{attribute addProperty BoxType "EPP3744-0041-0016"}
{attribute addProperty Id "Safe_State_ActiveAT %I*BOOL811Sync_errorAT %I*BOOL8114Undervoltage_UsAT %I*BOOL811Undervoltage_UpAT %I*BOOL812TxPDO_ToggleAT %I*BOOL8116"}
{attribute addProperty CRC "494286285"}
{attribute addProperty SizeInBites "40"}
{attribute addProperty SizeInBytes "5"}
TYPE DEV_Inputs_Device_1D7635CD :
STRUCT
	{attribute addProperty Name "Safe_State_Active"}
	Safe_State_Active AT %I* : BOOL;
	{attribute addProperty Name "Sync_error"}
	Sync_error AT %I* : BOOL;
	{attribute addProperty Name "Undervoltage_Us"}
	Undervoltage_Us AT %I* : BOOL;
	{attribute addProperty Name "Undervoltage_Up"}
	Undervoltage_Up AT %I* : BOOL;
	{attribute addProperty Name "TxPDO_Toggle"}
	TxPDO_Toggle AT %I* : BOOL;
END_STRUCT
END_TYPE

(* stored: Version 1.2.0.0, ProductVersion 3.1.4024.9
   DUT DEV_Inputs_Device_1D7635CD: Id {6080177e-ab39-4675-9a37-21fa589101b0} *)
